// TIA Portal V19 export
DATA_BLOCK "CoilHandling_PERS"   // DB73
// stored: MemoryReserve 100
   VAR RETAIN
      PersistentValues : "CoilHandling_Persistent";
   END_VAR
BEGIN
   PersistentValues.Data.MaterialPresence := TRUE;
   PersistentValues.Data.MaterialPresence_Decoiler := TRUE;
   PersistentValues.Data.MaterialPresence_StraightenerEntry := TRUE;
   PersistentValues.Data.MaterialPresence_StraightenerExit := TRUE;
   PersistentValues.Data.MaterialPresence_JBPinchExit := TRUE;
   PersistentValues.Data.MaterialPresence_RF_Entry := FALSE;
   PersistentValues.Data.MaterialFullLoaded := TRUE;
   PersistentValues.Data.VelocityOverride := 100.0;
   PersistentValues.Data.MATERIAL_SEPARATION.Mem := FALSE;
   PersistentValues.Data.MATERIAL_SEPARATION.CutDoneAndConfirmed := FALSE;
   PersistentValues.Data.END_OF_COIL.Mem := FALSE;
   PersistentValues.Data.END_OF_COIL.Tail_ReachCutPosition := FALSE;
   PersistentValues.Data.END_OF_COIL.Tail_CutDone := FALSE;
   PersistentValues.Data.END_OF_COIL.Tail_ReachJunctionPos := FALSE;
   PersistentValues.Data.END_OF_COIL.SaveEncPosAx_EndOfMaterialStraightEntry := 648210.821;
   PersistentValues.Data.END_OF_COIL.SaveEncPosAx_EndOfMaterialStraightExit := 649237.871;
   PersistentValues.Data.END_OF_COIL.SaveEncPosMat_CutDone := 655160.75488378;
   PersistentValues.Data.CoilLoadedInDecoiler1 := FALSE;
   PersistentValues.Data.CoilLoadedInDecoiler2 := FALSE;
   PersistentValues.Data.Thickness.Measure.BypassON := FALSE;
   PersistentValues.Data.Thickness.Measure.ID := 12;
   PersistentValues.Data.Thickness.Measure.Last_TriggerPosition := 676301.159149282;
   PersistentValues.Data.Thickness.Measure.AverageSum := 16.8089997768402;
   PersistentValues.Data.Thickness.Measure.OutOfRange_Counter := 0;
   PersistentValues.Data.Thickness.Measure.InRange_Counter := 12;
   PersistentValues.Data.Thickness.Measure.Buffer[1].ID := 12;
   PersistentValues.Data.Thickness.Measure.Buffer[2].ID := 11;
   PersistentValues.Data.Thickness.Measure.Buffer[3].ID := 10;
   PersistentValues.Data.Thickness.Measure.Buffer[4].ID := 9;
   PersistentValues.Data.Thickness.Measure.Buffer[5].ID := 8;
   PersistentValues.Data.Thickness.Measure.Buffer[6].ID := 7;
   PersistentValues.Data.Thickness.Measure.Buffer[7].ID := 6;
   PersistentValues.Data.Thickness.Measure.Buffer[8].ID := 5;
   PersistentValues.Data.Thickness.Measure.Buffer[9].ID := 4;
   PersistentValues.Data.Thickness.Measure.Buffer[10].ID := 3;
   PersistentValues.Data.Thickness.Measure.Buffer[1].Time_Stamp := DTL#2025-11-05-09:46:12.294572894;
   PersistentValues.Data.Thickness.Measure.Buffer[2].Time_Stamp := DTL#2025-11-05-09:42:47.882452468;
   PersistentValues.Data.Thickness.Measure.Buffer[3].Time_Stamp := DTL#2025-11-05-09:42:34.385550353;
   PersistentValues.Data.Thickness.Measure.Buffer[4].Time_Stamp := DTL#2025-11-05-09:42:30.186815230;
   PersistentValues.Data.Thickness.Measure.Buffer[5].Time_Stamp := DTL#2025-11-05-09:42:24.385450206;
   PersistentValues.Data.Thickness.Measure.Buffer[6].Time_Stamp := DTL#2025-11-05-09:42:18.218819246;
   PersistentValues.Data.Thickness.Measure.Buffer[7].Time_Stamp := DTL#2025-11-05-09:42:12.565298342;
   PersistentValues.Data.Thickness.Measure.Buffer[8].Time_Stamp := DTL#2025-11-05-09:42:07.877978702;
   PersistentValues.Data.Thickness.Measure.Buffer[9].Time_Stamp := DTL#2025-11-05-09:35:43.818079377;
   PersistentValues.Data.Thickness.Measure.Buffer[10].Time_Stamp := DTL#2025-11-05-09:34:12.274454908;
   PersistentValues.Data.Thickness.Measure.Buffer[1..10].Status := 1;
   PersistentValues.Data.Thickness.Measure.Buffer[1].Material_Position := 676301.159149282;
   PersistentValues.Data.Thickness.Measure.Buffer[2].Material_Position := 676001.023897475;
   PersistentValues.Data.Thickness.Measure.Buffer[3].Material_Position := 675700.998766472;
   PersistentValues.Data.Thickness.Measure.Buffer[4].Material_Position := 675400.573196182;
   PersistentValues.Data.Thickness.Measure.Buffer[5].Material_Position := 675100.565083848;
   PersistentValues.Data.Thickness.Measure.Buffer[6].Material_Position := 674800.397796898;
   PersistentValues.Data.Thickness.Measure.Buffer[7].Material_Position := 674500.198474805;
   PersistentValues.Data.Thickness.Measure.Buffer[8].Material_Position := 674199.962112077;
   PersistentValues.Data.Thickness.Measure.Buffer[9].Material_Position := 673899.909951422;
   PersistentValues.Data.Thickness.Measure.Buffer[10].Material_Position := 673599.901839088;
   PersistentValues.Data.Thickness.Measure.Buffer[1].Value := 1.524;
   PersistentValues.Data.Thickness.Measure.Buffer[2].Value := 1.532;
   PersistentValues.Data.Thickness.Measure.Buffer[3].Value := 1.518;
   PersistentValues.Data.Thickness.Measure.Buffer[4].Value := 1.517;
   PersistentValues.Data.Thickness.Measure.Buffer[5].Value := 1.532;
   PersistentValues.Data.Thickness.Measure.Buffer[6].Value := 1.516;
   PersistentValues.Data.Thickness.Measure.Buffer[7].Value := 1.535;
   PersistentValues.Data.Thickness.Measure.Buffer[8].Value := 1.537;
   PersistentValues.Data.Thickness.Measure.Buffer[9].Value := 1.548;
   PersistentValues.Data.Thickness.Measure.Buffer[10].Value := 1.513;
   PersistentValues.Data.Thickness.Measure.Buffer[1].Err := 0.02400005;
   PersistentValues.Data.Thickness.Measure.Buffer[2].Err := 0.03199995;
   PersistentValues.Data.Thickness.Measure.Buffer[3].Err := 0.01800001;
   PersistentValues.Data.Thickness.Measure.Buffer[4].Err := 0.01699996;
   PersistentValues.Data.Thickness.Measure.Buffer[5].Err := 0.03199995;
   PersistentValues.Data.Thickness.Measure.Buffer[6].Err := 0.01600003;
   PersistentValues.Data.Thickness.Measure.Buffer[7].Err := 0.03499997;
   PersistentValues.Data.Thickness.Measure.Buffer[8].Err := 0.03699994;
   PersistentValues.Data.Thickness.Measure.Buffer[9].Err := 0.04799998;
   PersistentValues.Data.Thickness.Measure.Buffer[10].Err := 0.01300001;
   PersistentValues.Data.Thickness.Measure.Buffer[1].Avg := 1.528091;
   PersistentValues.Data.Thickness.Measure.Buffer[2].Avg := 1.527454;
   PersistentValues.Data.Thickness.Measure.Buffer[3].Avg := 1.527;
   PersistentValues.Data.Thickness.Measure.Buffer[4].Avg := 1.528;
   PersistentValues.Data.Thickness.Measure.Buffer[5].Avg := 1.529375;
   PersistentValues.Data.Thickness.Measure.Buffer[6].Avg := 1.529;
   PersistentValues.Data.Thickness.Measure.Buffer[7].Avg := 1.531167;
   PersistentValues.Data.Thickness.Measure.Buffer[8].Avg := 1.5304;
   PersistentValues.Data.Thickness.Measure.Buffer[9].Avg := 1.52875;
   PersistentValues.Data.Thickness.Measure.Buffer[10].Avg := 1.522333;
   PersistentValues.Data.Thickness.Measure.Buffer[1].AvgErr := 0.02809083;
   PersistentValues.Data.Thickness.Measure.Buffer[2].AvgErr := 0.0274545;
   PersistentValues.Data.Thickness.Measure.Buffer[3].AvgErr := 0.02699995;
   PersistentValues.Data.Thickness.Measure.Buffer[4].AvgErr := 0.028;
   PersistentValues.Data.Thickness.Measure.Buffer[5].AvgErr := 0.02937496;
   PersistentValues.Data.Thickness.Measure.Buffer[6].AvgErr := 0.02899992;
   PersistentValues.Data.Thickness.Measure.Buffer[7].AvgErr := 0.03116667;
   PersistentValues.Data.Thickness.Measure.Buffer[8].AvgErr := 0.03039992;
   PersistentValues.Data.Thickness.Measure.Buffer[9].AvgErr := 0.02874994;
   PersistentValues.Data.Thickness.Measure.Buffer[10].AvgErr := 0.02233326;
   PersistentValues.Data.Thickness.MES_Record.ID := 12;
   PersistentValues.Data.Thickness.MES_Record.Time_Stamp := DTL#2025-11-05-09:46:12.294572894;
   PersistentValues.Data.Thickness.MES_Record.Status := 1;
   PersistentValues.Data.Thickness.MES_Record.Material_Position := 676301.159149282;
   PersistentValues.Data.Thickness.MES_Record.Value := 1.524;
   PersistentValues.Data.Thickness.MES_Record.Err := 0.02400005;
   PersistentValues.Data.Thickness.MES_Record.Avg := 1.528091;
   PersistentValues.Data.Thickness.MES_Record.AvgErr := 0.02809083;
   PersistentValues.Par.MaterialBkw_PercentageStraightener := 5.0;
   PersistentValues.Par.ExtraLowSpeed_Percentage := 10.0;
   PersistentValues.Par.TimeStopInactivity := T#5M;
   PersistentValues.Par.SemiAut.Vel_Fwd := 6000.0;
   PersistentValues.Par.SemiAut.Vel_Bkw := 6000.0;
   PersistentValues.Par.SemiAut.Acc := 1000.0;
   PersistentValues.Par.SemiAut.Dec := 1000.0;
   PersistentValues.Par.SemiAut.Jerk := 10000.0;
   PersistentValues.Par.CoilEnd.EnableCoilTailSequence := TRUE;
   PersistentValues.Par.CoilEnd.Distance_StraightEntry_To_StraightExit := 300.0;
   PersistentValues.Par.CoilEnd.Distance_StraightEntry_To_CutExecution := 400.0;
   PersistentValues.Par.CoilEnd.Distance_StraightEntry_to_JunctionExecution := 401.0;
   PersistentValues.Par.CoilEnd.Distance_CutHead_to_JB := 810.0;
   PersistentValues.Par.CoilEnd.Tol_CheckSensorStraightExit := 1.0;
   PersistentValues.Par.CoilEnd.Tol_PosCutExecution := 1.0;
   PersistentValues.Par.CoilEnd.Tol_PosJunctionExecution := 1.0;
   PersistentValues.Par.CoilEnd.Delay_PinchrollFwd := T#0MS;
   PersistentValues.Par.CoilEnd.Delay_StraightnerBwd := T#10S;
   PersistentValues.Par.CoilEnd.Vel := 3000.0;
   PersistentValues.Par.CoilEnd.Acc := 1000.0;
   PersistentValues.Par.CoilEnd.Dec := 1000.0;
   PersistentValues.Par.CoilEnd.Jerk := 10000.0;
   PersistentValues.Par.CoilEnd.PercentageStraightener := 5.0;
   PersistentValues.Par.Thickness.SensorON := TRUE;
   PersistentValues.Par.Thickness.Trigger_interval := 300.0;
   PersistentValues.Par.Thickness.NG_Measures_ToFault := 10;
   PersistentValues.Par.Thickness.BypassAutoReset := 5;
   PersistentValues.Par.Thickness.Tolerance_Min := -0.2;
   PersistentValues.Par.Thickness.Tolerance_Max := 0.2;
   PersistentValues.Par.Thickness.MES_RecordChange_ThresholdMin := -0.05;
   PersistentValues.Par.Thickness.MES_RecordChange_ThresholdMax := 0.05;
END_DATA_BLOCK
